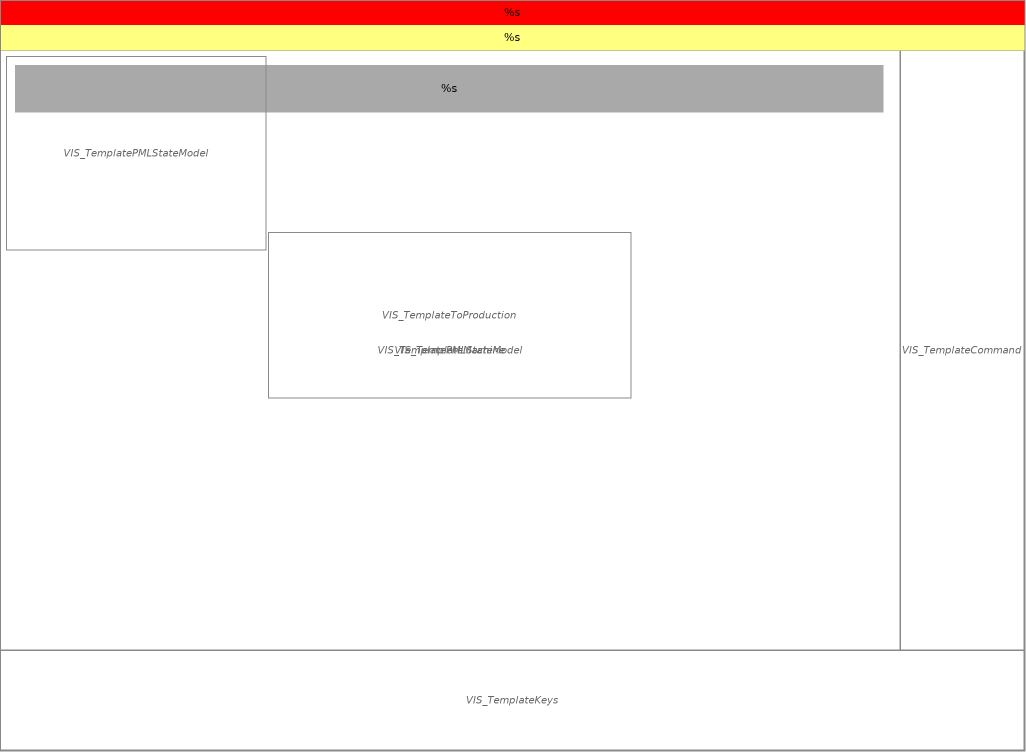
VISUALIZATION VIS_Main  // 1026x752
    Frame (0,50 900x600), invisible if: MAIN.fbVisu.iFrameVisible = 0 OR MAIN.fbMachine.bChangeIntoProduction
        shows VIS_TemplatePMLStateModel(ePMLUnitMode := MAIN.fbVisu.eModeVisu, ePMLState := MAIN.fbVisu.eStateVisu)
    Frame (268,232 363x166), invisible if: NOT MAIN.fbMachine.bChangeIntoProduction
        shows VIS_TemplateToProduction(stChangeIntoProduction := stChangeIntoProduction)
    Textfield (15,65 868x47), "%s", text variable: MAIN.fbVisu.sUnitName, invisible if: MAIN.fbVisu.iFrameVisible = 0 OR MAIN.fbMachine.bChangeIntoProduction
    Frame (0,50 900x600), invisible if: MAIN.fbVisu.iFrameVisible > 0 OR MAIN.fbMachine.bChangeIntoProduction
        shows VIS_TemplateMachine()
    Rectangle (0,0 1024x25), "%s", text variable: MAIN.fbVisu.sAlarmVisu, invisible if: (MAIN.fbMachine.bChangeIntoProduction OR MAIN.fbVisu.sAlarmVisu = '')
    Frame (900,50 124x600)
        shows VIS_TemplateCommand(eModeCommand := PackTags.Command.UnitMode, eStateCommand := PackTags.Command.CntrlCmd, eModeStatus := PackTags.Status.UnitModeCurrent, eStateStatus := PackTags.Status.StateCurrent, bModeChangeReq := PackTags.Command.UnitModeChangeRequest)
    Frame (0,650 1024x100)
        shows VIS_TemplateKeys(Caption := aCaption, KeyPressed := aKeyPressed)
    Frame (6,56 260x194), invisible if: MAIN.fbVisu.iFrameVisible > 0 OR MAIN.fbMachine.bChangeIntoProduction
        shows VIS_TemplatePMLStateModel(ePMLUnitMode := PackTags.Status.UnitModeCurrent, ePMLState := PackTags.Status.StateCurrent)
    Rectangle (0,25 1024x25), "%s", text variable: MAIN.fbVisu.sWarningVisu, invisible if: (MAIN.fbMachine.bChangeIntoProduction OR MAIN.fbVisu.sWarningVisu ='')
END_VISUALIZATION

(* stored: Version 1.1.0.1
   Visu VIS_Main: Id {e1801763-8c99-49e1-8dd6-d8ae8e1af5ae} *)
